TYPE MC_CAM_REF :
STRUCT
END_STRUCT
END_TYPE

(* stored: Version 1.1.0.1, ProductVersion 3.1.4024.11
   DUT MC_CAM_REF: Id {3eef7930-775f-40e4-a459-1ef36912170f} *)
